// TIA Portal V18 export
// export: Created 2026-03-12T16:04:35.6703983Z, ExportSetting WithDefaults, DisplayName Totally Integrated Automation Portal, DisplayVersion V18 Update 5, DisplayName TIA Portal Openness, DisplayVersion V18 Update 5, DisplayName TIA Portal Version Control Interface, DisplayVersion V18, DisplayName SINAMICS Startdrive Advanced, DisplayVersion V18, DisplayName SINAMICS Startdrive G130, G150, S120, S150, SINAMICS MV, S210, DisplayVersion V18, DisplayName SINAMICS Startdrive G110M, G120, G120C, G120D, G120P, G115D, DisplayVersion V18, DisplayName STEP 7 Professional, DisplayVersion V18 Update 5, DisplayName STEP 7 Safety, DisplayVersion V18, DisplayName WinCC Professional, DisplayVersion V18 Update 5
FUNCTION_BLOCK "FB_Gateway_MK5_Driver"   // FB30, SCL
{ S7_Optimized_Access := 'TRUE' }
VERSION : 0.1
// stored: AutoNumber true, IsIECCheckEnabled false, IsRetainMemResEnabled false, MemoryReserve 100, SetENOAutomatically false, UDAEnableTagReadback false
   VAR_INPUT
      Enable : Bool;
      NodeID_Start : Byte;   // Endereço do dispositivo
      NodeID_End : Byte;
      NumVars : Int;   // Quantidade de parâmetros a ler (1..8)
      ParamList : Array[1..8] of Int;   // Lista de parametros ID's
   END_VAR
   VAR_OUTPUT
      Busy : Bool;
      Done : Bool;
      CurrentNode : Byte;
      Error : Bool;
      Buffer_Var_Out : Array[1..8] of DWord;
   END_VAR
   VAR_IN_OUT
      Header_In : "Header";
      Buffer_In : "Buff_64";
      Header_Out : "Header";
      Buffer_Out : "Buff_64";
   END_VAR
   VAR
      State : Int;
      SyncToggle : Bool;
      NodeID_Current : Byte;
      i : Int;
      ParamWord : Word;
   END_VAR
BEGIN
   CASE #State OF

           //-------------------------------------------------
       0: // IDLE
           //-------------------------------------------------
           #Done := FALSE;
           #Busy := FALSE;

           IF #Enable THEN
               #NodeID_Current := #NodeID_Start;
               #CurrentNode := #NodeID_Current;
               #Busy := TRUE;
               #State := 1;
           END_IF;


           //-------------------------------------------------
       1: // BUILD FRAME
           //-------------------------------------------------

           // Alterna Sync
           #SyncToggle := NOT #SyncToggle;

           #Header_Out.Sync_bit_6 := #SyncToggle;
           #Header_Out.Sync_bit_7 := FALSE;

           // Função READ = 001
           #Header_Out.Function_bit_3 := TRUE;
           #Header_Out.Function_bit_4 := FALSE;
           #Header_Out.Function_bit_5 := FALSE;

           // Número de registros
           #Header_Out.Param_bit_0 := (#NumVars AND 1) <> 0;
           #Header_Out.Param_bit_1 := (#NumVars AND 2) <> 0;
           #Header_Out.Param_bit_2 := (#NumVars AND 4) <> 0;

           // Limpa buffer
           FOR #i := 1 TO 8 DO
               #Buffer_Out.Buffer[#i].Node := 0;
               #Buffer_Out.Buffer[#i].Param_MSB := 0;
               #Buffer_Out.Buffer[#i].Param_LSB := 0;
               #Buffer_Out.Buffer[#i].Data_1 := 0;
               #Buffer_Out.Buffer[#i].Data_2 := 0;
               #Buffer_Out.Buffer[#i].Data_3 := 0;
               #Buffer_Out.Buffer[#i].Data_4 := 0;
           END_FOR;

           // Preenche registros para este Node
           FOR #i := 1 TO #NumVars DO

               #ParamWord := INT_TO_WORD(#ParamList[#i]);

               #Buffer_Out.Buffer[#i].Node := #NodeID_Current;

               #Buffer_Out.Buffer[#i].Param_MSB := WORD_TO_BYTE(SHR(IN := #ParamWord,N:= 8));

               #Buffer_Out.Buffer[#i].Param_LSB := WORD_TO_BYTE(#ParamWord);

           END_FOR;

           #State := 2;


           //-------------------------------------------------
       2: // WAIT RESPONSE
           //-------------------------------------------------

           // Aguarda Sync refletido no Header de entrada
           IF #Header_In.Sync_bit_6 = #SyncToggle  AND #Header_In.Sync_bit_7 = FALSE   THEN

               // Leitura concluída para este Node

               FOR #i := 1 TO 8 DO

                   #Buffer_Var_Out[#i] :=
                               BYTE_TO_DWORD(#Buffer_In.Buffer[#i].Data_1) OR
                   SHL(IN :=   BYTE_TO_DWORD(#Buffer_In.Buffer[#i].Data_2), N := 8 ) OR
                   SHL(IN :=   BYTE_TO_DWORD(#Buffer_In.Buffer[#i].Data_3), N := 16) OR
                   SHL(IN :=   BYTE_TO_DWORD(#Buffer_In.Buffer[#i].Data_4), N := 24);

               END_FOR;

               IF #NodeID_Current < #NodeID_End THEN

                   #NodeID_Current := #NodeID_Current + 1;
                   #CurrentNode := #NodeID_Current;
                   #State := 1;     // próximo soprador

               ELSE

                   #Done := TRUE;
                   #Busy := FALSE;
                   #State := 0;

               END_IF;

           END_IF;

   END_CASE;
END_FUNCTION_BLOCK
